FUNCTION FIELDBUS_WORD_TO_PERCENT (* Convert a REAL in the Range 0.0 to 100.0 to a WORD Value Range 0-FAFF *)
  (* Standard: SAE J1939; ISO 11783; Description: Copyright (c) 2023 HR Agrartechnik GmbH This program and the accompanying materials are made available under the terms of the Eclipse Public License 2.0 which is available at https://www.eclipse.org/legal/epl-2.0/ SPDX-License-Identifier: EPL-2.0 *)
  (* Version 1.0, 2023-10-21, Franz Höpfinger, HR Agrartechnik GmbH *)
  (* Version 1.1, 2024-09-19, Franz Höpfinger, HR Agrartechnik GmbH, Update to a more Function like Interface *)
  PACKAGE signalprocessing;
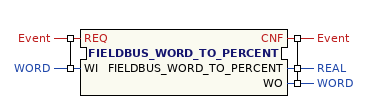
  EVENT_INPUT
    REQ WITH WI;
  END_EVENT
  EVENT_OUTPUT
    CNF WITH FIELDBUS_WORD_TO_PERCENT, WO;
  END_EVENT
  VAR_INPUT
    WI : WORD; (* Input Value *)
  END_VAR
  VAR_OUTPUT
    FIELDBUS_WORD_TO_PERCENT : REAL;
    WO : WORD; (* Input Value mirror if Signal Valid. *)
  END_VAR
  BODY IN ST:
PACKAGE signalprocessing;

(* Convert a REAL in the Range 0.0 to 100.0 to a WORD Value Range 0-FAFF *)
FUNCTION FIELDBUS_WORD_TO_PERCENT : REAL
VAR_INPUT
	WI : WORD; // Input Value
END_VAR

VAR_OUTPUT
	WO : WORD; // Input Value mirror if Signal Valid.
END_VAR

IF (WI <= FIELDBUS_SIGNAL::VALID_SIGNAL_W) THEN
	WO := WI;
	FIELDBUS_WORD_TO_PERCENT := UDINT_TO_REAL(WORD_TO_UDINT(WO))
		/ UDINT_TO_REAL(WORD_TO_UDINT(FIELDBUS_SIGNAL::VALID_SIGNAL_W));
END_IF;

END_FUNCTION
  END_BODY
END_FUNCTION
